PROGRAM MAIN
VAR
	//Time Function Blocks
	fbGetTimeZone : FB_GetTimeZoneInformation;
	fb_Get_LocTime : FB_LocalSystemTime;
	fb_LocTime_to_UTC : FB_TzSpecificLocalTimeToSystemTime;
	//fb_UTC_to_LocTime : FB_SystemTimeToTzSpecificLocalTime;
	
	//Timer Function Block
    logTimer : TON := ( IN := TRUE, PT := T#500MS );	
	
END_VAR

//Start of the PLC Code
(*

IN ORDER TO USE THESE FUNCTION BLOCKS, YOU NEED TO INSTALL THE Tc2_Utilities LIBRARY

The Outputs of the TzSpecific Function blocks is a TIMESTRUCT. 

FB_LocalSystemTime:
This function block internally combines the functions of the following function blocks: RTC_EX2, NT_GetTime, FB_GetTimeZoneInformation and NT_SetTimeToRTCTime. 
The FB_LocalSystemTime function block must be called cyclically (e.g. every second or during each PLC cycle). This is necessary to enable the time between synchronizations to be calculated.
 - sNetID  : Can use AMS id of a target computer, for Local Computer = empty string ''
 - dwCycle : When the FB resynchronize its local time w/ the system time default is 5 sec

FB_TzSpecificLocalTimeToSystemTime:
	TzSpecificLocalTime = LocalSystemTime
	SystemTime = Cordinated Universal Time (UTC)



*)

//Get Time Zone information. This is used when converting UTC to Local Time
fbGetTimeZone(
	sNetID:='' , 
	bExecute:= TRUE, 
	tTimeout:= , 
	bBusy=> , 
	bError=> , 
	nErrID=> , 
	tzID=> , 
	tzInfo=> );

// Get Local Time
fb_Get_LocTime(
	sNetID:= '', 
	bEnable:= TRUE, 
	dwCycle:= 1, 
	dwOpt:= , 
	tTimeout:= , 
	bValid=> , 
	systemTime=> , 
	tzID=> );

 // Valid Time to convert
IF fb_Get_LocTime.bValid THEN
	
	//Convert to UTC. in : Local Time, tzInfo : The timezone you're in
	fb_LocTime_to_UTC(
	in:= fb_Get_LocTime.systemTime, 
	tzInfo:= fbGetTimeZone.tzInfo, 
	out=> , 
	eTzID=> , 
	bB=> );
  
END_IF

(* 
	//Convert from UTC time to Local Time
	fb_UTC_to_LocTime(
	in:= fb_LocTime_to_UTC.out, 
	tzInfo:= fbGetTimeZone.tzInfo, 
	out=> , 
	eTzID=> , 
	bB=> );
*)

//Timer for displaying times	
logTimer( IN := fb_Get_LocTime.bValid );
IF logTimer.Q THEN
	logTimer( IN := FALSE ); logTimer( IN := fb_Get_LocTime.bValid );
	ADSLOGSTR( ADSLOG_MSGTYPE_HINT OR ADSLOG_MSGTYPE_LOG, 'Local Time:	%s', SYSTEMTIME_TO_STRING(fb_Get_LocTime.systemTime));
	ADSLOGSTR( ADSLOG_MSGTYPE_HINT OR ADSLOG_MSGTYPE_LOG, 'UTC Time:	%s', SYSTEMTIME_TO_STRING(fb_LocTime_to_UTC.out));
END_IF

END_PROGRAM

(* stored: Version 1.1.0.1, ProductVersion 3.1.4024.12
   POU MAIN: Id {c9cfe12a-66bd-4ab5-be78-11604f09586a}, SpecialFunc None *)
